// TIA Portal V16 export
// export: Created 2019-09-22T11:06:10.7517431Z, ExportSetting WithDefaults, DisplayName Totally Integrated Automation Portal, DisplayVersion V16, DisplayName TIA Portal Version Control Interface, DisplayVersion V16, DisplayName TIA Portal Openness, DisplayVersion V16, DisplayName STEP 7 Professional, DisplayVersion V16, DisplayName SIMATIC Energy Suite, DisplayVersion V16, DisplayName STEP 7 Safety, DisplayVersion V16, DisplayName WinCC Professional, DisplayVersion V16, DisplayName SIMATIC Visualization Architect, DisplayVersion V16
TYPE "typeShowDevice"
// stored: IsFailsafeCompliant false
   STRUCT
      stationNumber : UInt;   // Station Number of interfaces in HW configuration
      "name" : String[50];   // Device name
      errorState : USInt;   // Status of the device 1=ok!, 2=faulty, 3=lost connection, 4=disabled, 12= was faulty, 13=was lost, 14=was disabled
      slot { S7_SetPoint := 'True'} : Array[0.."MAX_MODULES_DEVICE"] of "typeShowModul";   // slot informations
   END_STRUCT;
END_TYPE
